// TIA Portal project "Egzamin zawodowy czerwiec 2013" (V11)

(* hardware
DEVICE "S7-400 station_1"  S7400.Device
   slot 0: "UR1_0"  UR1  6ES7 400-1TA01-0AA0
   slot 2: "PLC_1"  CPU 416F-3 PN/DP  6ES7 416-3FR05-0AB0  V5.3
      slot 5: "PROFINET interface_1"  PN-IO
         slot 1: "Port_1"  Port
         slot 2: "Port_2"  Port
*)

// ===== PLC "PLC_1"  CPU 416F-3 PN/DP =====

VAR_GLOBAL   // PLC tag table "Default tag table"
   "S1" AT %I0.0 : Bool;
   "B2" AT %I0.1 : Bool;
   "ruch dół" AT %M0.0 : Bool;
   "Tag_1" AT %M1.0 : Bool;
   "Tag_2" AT %T1 : Timer;
   "miganie lampki" AT %M0.1 : Bool;
   "zawór" AT %Q0.0 : Bool;
   "b1" AT %I0.2 : Bool;
   "głowica na dole" AT %M0.2 : Bool;
   "zgrzewanie" AT %M0.3 : Bool;
   "lampka" AT %Q0.3 : Bool;
   "stop grzania" AT %M0.5 : Bool;
   "grzanie" AT %Q0.2 : Bool;
   "grzanie(1)" AT %Q0.1 : Bool;
END_VAR

ORGANIZATION_BLOCK "Main"   // OB1, LAD
TITLE = "Main Program Sweep (Cycle)"
{ S7_Optimized_Access := 'FALSE' }
VERSION : 0.1
   VAR_TEMP
      OB1_EV_CLASS : Byte;   // Bits 0-3 = 1 (Coming event), Bits 4-7 = 1 (Event class 1)
      OB1_SCAN_1 : Byte;   // 1 (Cold restart scan 1 of OB 1), 3 (Scan 2-n of OB 1)
      OB1_PRIORITY : Byte;   // Priority of OB Execution
      OB1_OB_NUMBR : Byte;   // 1 (Organization block 1, OB1)
      OB1_RESERVED_1 : Byte;   // Reserved for system
      OB1_RESERVED_2 : Byte;   // Reserved for system
      OB1_PREV_CYCLE : Int;   // Cycle time of previous OB1 scan (milliseconds)
      OB1_MIN_CYCLE : Int;   // Minimum cycle time of OB1 (milliseconds)
      OB1_MAX_CYCLE : Int;   // Maximum cycle time of OB1 (milliseconds)
      OB1_DATE_TIME : Date_And_Time;   // Date and time OB1 started
   END_VAR
   VAR_TEMP   // added for the SCL form of the ladder/FBD networks
      _w1 : Bool;
      _s5time1 : S5Time;
   END_VAR
BEGIN

REGION Network 1
   // Wciśnięty S1 i pozycja góra B2 - rozpoczyna ruch w dół
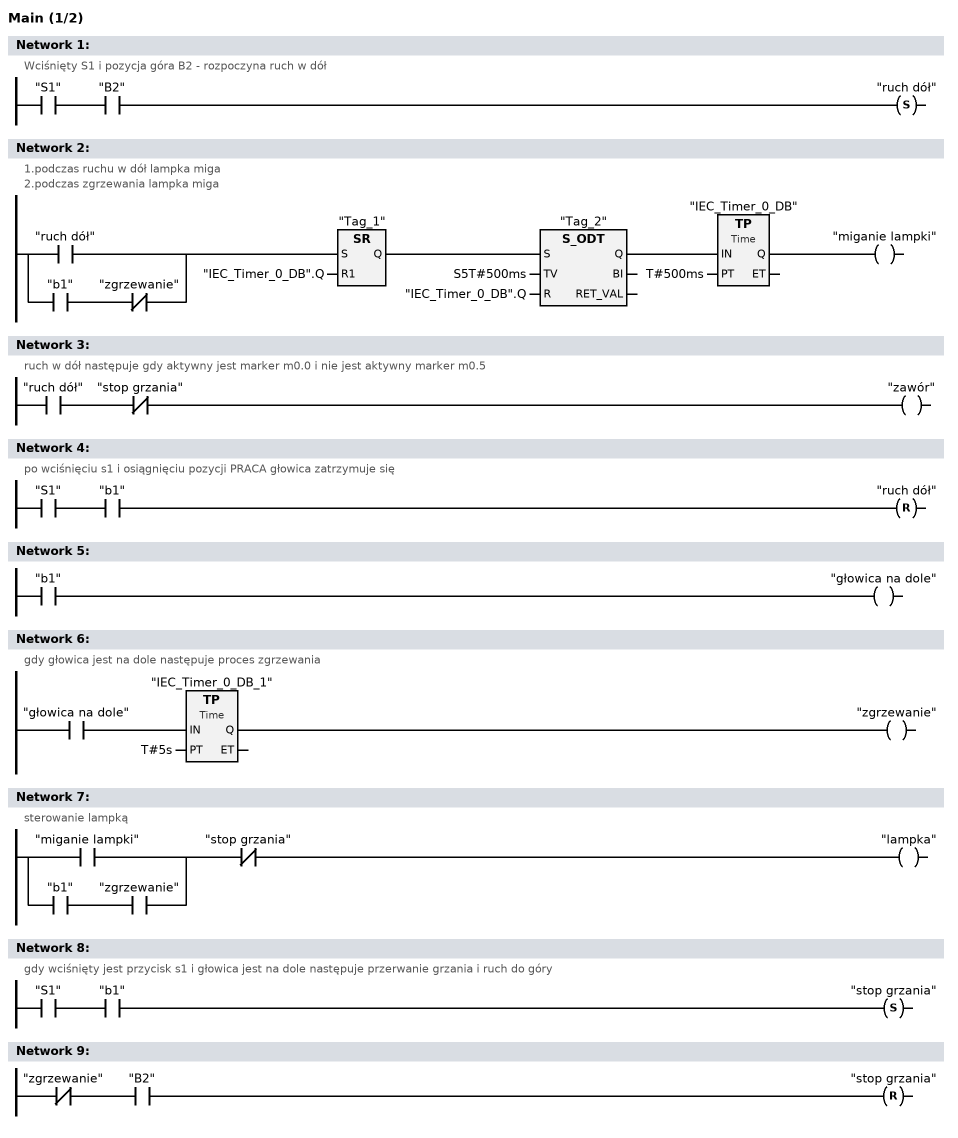
   RUNG wire#powerrail
      Contact( "S1" )
      Contact( "B2" )
      S_Coil( "ruch dół" )
   END_RUNG
   // the same network as SCL:
   IF "S1" AND "B2" THEN "ruch dół" := TRUE; END_IF;
END_REGION

REGION Network 2
   // 1.podczas ruchu w dół lampka miga
   // 2.podczas zgrzewania lampka miga
   IF "ruch dół" OR ("b1" AND NOT "zgrzewanie") THEN
       "Tag_1" := TRUE;   // SR flip-flop
   END_IF;
   IF "IEC_Timer_0_DB".Q THEN "Tag_1" := FALSE; END_IF;
   #_s5time1 := S_ODT(T_NO := "Tag_2", S := "Tag_1", TV := S5T#500ms, R := "IEC_Timer_0_DB".Q, Q => #_w1);
   "IEC_Timer_0_DB".TP(IN := #_w1, PT := T#500ms);
   "miganie lampki" := "IEC_Timer_0_DB".Q;
END_REGION

REGION Network 3
   // ruch w dół następuje gdy aktywny jest marker m0.0 i nie jest aktywny marker m0.5
   RUNG wire#powerrail
      Contact( "ruch dół" )
      I_Contact( "stop grzania" )
      Coil( "zawór" )
   END_RUNG
   // the same network as SCL:
   "zawór" := "ruch dół" AND NOT "stop grzania";
END_REGION

REGION Network 4
   // po wciśnięciu s1 i osiągnięciu pozycji PRACA głowica zatrzymuje się
   RUNG wire#powerrail
      Contact( "S1" )
      Contact( "b1" )
      R_Coil( "ruch dół" )
   END_RUNG
   // the same network as SCL:
   IF "S1" AND "b1" THEN "ruch dół" := FALSE; END_IF;
END_REGION

REGION Network 5
   RUNG wire#powerrail
      Contact( "b1" )
      Coil( "głowica na dole" )
   END_RUNG
   // the same network as SCL:
   "głowica na dole" := "b1";
END_REGION

REGION Network 6
   // gdy głowica jest na dole następuje proces zgrzewania
   "IEC_Timer_0_DB_1".TP(IN := "głowica na dole", PT := T#5s);
   "zgrzewanie" := "IEC_Timer_0_DB_1".Q;
END_REGION

REGION Network 7
   // sterowanie lampką
   RUNG wire#powerrail
      Contact( "miganie lampki" )
      wire#w1
      I_Contact( "stop grzania" )
      Coil( "lampka" )
   END_RUNG
   RUNG wire#powerrail
      Contact( "b1" )
      Contact( "zgrzewanie" )
   END_RUNG wire#w1
   // the same network as SCL:
   "lampka" := ("miganie lampki" OR ("b1" AND "zgrzewanie")) AND NOT "stop grzania";
END_REGION

REGION Network 8
   // gdy wciśnięty jest przycisk s1 i głowica jest na dole następuje przerwanie grzania i ruch do góry
   RUNG wire#powerrail
      Contact( "S1" )
      Contact( "b1" )
      S_Coil( "stop grzania" )
   END_RUNG
   // the same network as SCL:
   IF "S1" AND "b1" THEN "stop grzania" := TRUE; END_IF;
END_REGION

REGION Network 9
   RUNG wire#powerrail
      I_Contact( "zgrzewanie" )
      Contact( "B2" )
      R_Coil( "stop grzania" )
   END_RUNG
   // the same network as SCL:
   IF NOT "zgrzewanie" AND "B2" THEN "stop grzania" := FALSE; END_IF;
END_REGION

REGION Network 10
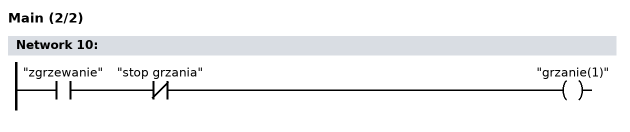
   RUNG wire#powerrail
      Contact( "zgrzewanie" )
      I_Contact( "stop grzania" )
      Coil( "grzanie(1)" )
   END_RUNG
   // the same network as SCL:
   "grzanie(1)" := "zgrzewanie" AND NOT "stop grzania";
END_REGION
END_ORGANIZATION_BLOCK